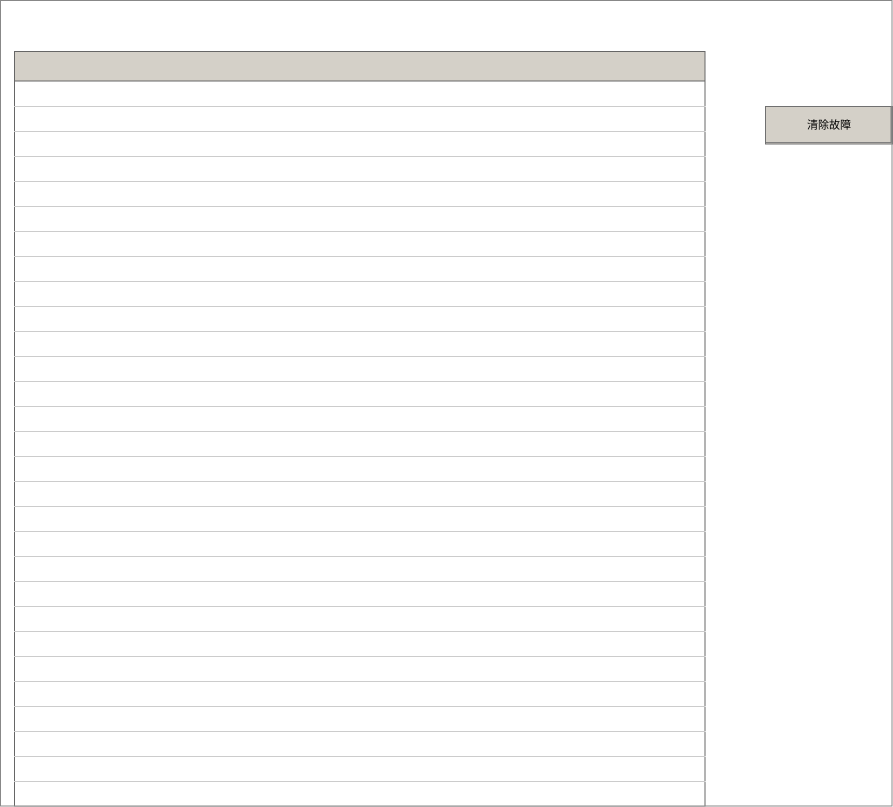
VISUALIZATION arm1SafetyCheck  // 893x807
    Table (14,51 691x756), data array: g_ArrayErrCodeTypeTest[1]
        p3854506369: g_ArrayErrCodeTypeTest[1][1][INDEX]
        p1892666644: g_ArrayErrCodeTypeTest[1][2][INDEX]
        p338671338: g_ArrayErrCodeTypeTest[3][INDEX]
        p2170511999: g_ArrayErrCodeTypeTest[4][INDEX]
        p3723444502: g_ArrayErrCodeTypeTest[5][INDEX]
    Button (765,106 128x38), "清除故障", colour toggle: g_clearFault
        tap g_clearFault
END_VISUALIZATION

(* stored: Version 1.1.0.1, ProductVersion 3.1.4024.11
   Visu arm1SafetyCheck: Id {301e62c0-83de-45da-b204-533c8e74a1cd} *)
